# EPICS autosave request: stdApp/Db/genericStateAux_settings.req
$(P)$(S)$(G)mode.VAL
$(P)$(S)$(G)desc.VAL
